PROGRAM MAIN
VAR
	//A4
	myWord : WORD := 16#5D7A;
	myWord2 : WORD;
	//A5
	myDWord : DWORD := 16#5D7A;
	myDWord2 : DWORD;
	myWord3 : WORD := 2#1111000011110000;
	
	//A7
	myRealArray: ARRAY[0..9] OF REAL := [1.1, 2.2, 3.3, 4.4, 5.5,6.6,7.7,8.8,9.9,10.10];  // Array mit 10 Elementen vom Typ REAL
	
	//A8
	index: INT;
	sum: REAL;
	mult: REAL;
	
	//A11
	bTasterblau : BOOL := TRUE;
	bTastergelb : BOOL := TRUE;
	blue_been_pressed : BOOL := FALSE;
	blue_led : BOOL := FALSE;
	blue_Counter : uint := 0;
	uiNumberPositiveEdgeBlue : UINT := 0;
	blueEdgeDetector : FB_EdgeDetector;
	yellowEdgeDetector : FB_EdgeDetector;
	
	//A14
	bufferArray : ARRAY[0..99] OF REAL ;
	
	
END_VAR

//frage wie kann man LED ansteueren?
//frage Ausgabe UltracSonic senosr?

//A4
myWord2 := SHR(myWord,3);
myDWord2 := SHL(myDWord,3);

//A5
myDWord2 := myWord OR 16#F0000000;

//A6
F_A06(16#1D06);

//A8
sum := 0;
mult := 1;
FOR index := 0 TO 9 DO
    sum := sum + myRealArray[index];  // Addiere den Schleifenindex zur Summe
	mult := mult * myRealArray[index];  // Addiere den Schleifenindex zur Summe
END_FOR;

//A9
sum := 0;
mult := 1;
index := 0;
WHILE index < 10 DO
	sum := sum + myRealArray[index];  // Addiere den Schleifenindex zur Summe
	mult := mult * myRealArray[index];  // Addiere den Schleifenindex zur Summe
	index := index +1;
END_WHILE;

//A10
index := 0;
REPEAT
    sum := sum + myRealArray[index];  // Addiere den Schleifenindex zur Summe
	mult := mult * myRealArray[index];  // Addiere den Schleifenindex zur Summe
	index := index +1;
UNTIL index < 10
END_REPEAT;

//A11
blueEdgeDetector(inputValue := bTasterblau, DoublePressedTime := 5);
IF blueEdgeDetector.risingEdge = TRUE THEN
	uiNumberPositiveEdgeBlue := uiNumberPositiveEdgeBlue + 1;
	
	//A12
	blue_been_pressed := NOT blue_been_pressed;
	blue_Counter := 0;
END_IF
yellowEdgeDetector(inputValue := bTastergelb, DoublePressedTime := 10);

//12
IF blue_been_pressed = TRUE THEN
	blue_Counter := blue_Counter + 1;
	IF blue_Counter >= 33 THEN
		blue_led := NOT blue_led;
		blue_Counter := 0;
	END_IF
END_IF

//A14
shiftLeft(bufferArray);
averageCalculator(bufferArray);

END_PROGRAM

(* stored: Version 1.1.0.1, ProductVersion 3.1.4024.13
   POU MAIN: Id {931ab9aa-2266-4aee-b72b-9592c3769ea8}, SpecialFunc None *)
